RoboDK station: GenerischV4_OPCUA_cubestation.rdk

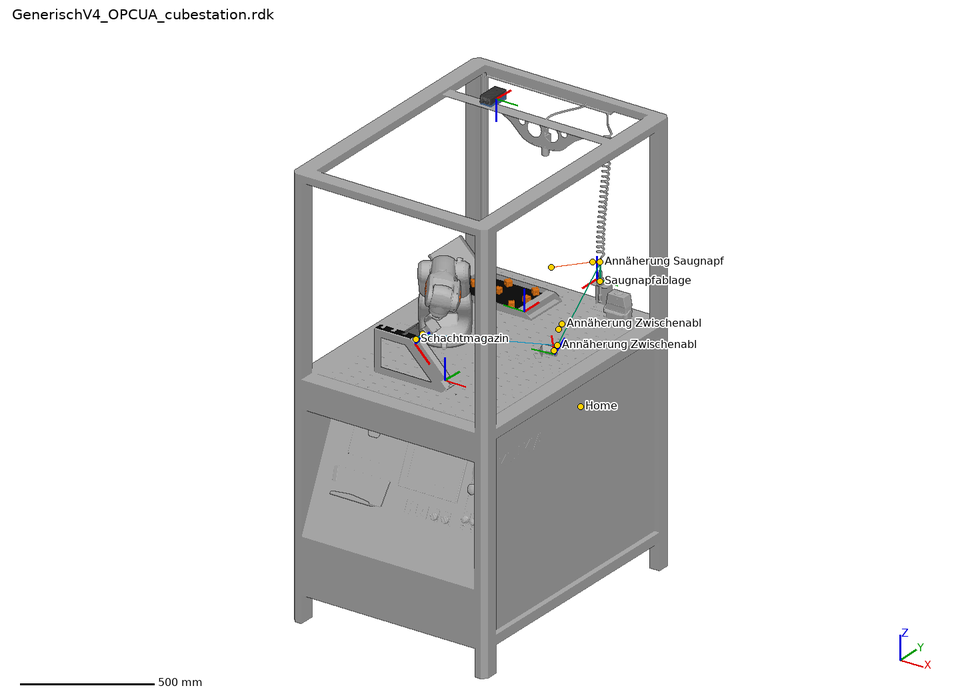
[picture v0: the station drawn from its stored meshes, robots at their saved joint values, targets as dots, program paths as lines]
Station GenerischV4_cubestation (saved by RoboDK 5.9.4). Poses are relative to the parent item; angles as X-Y-Z fixed-axis rotations.
Station parameters (name, value as stored): CMD_Objektposition, 0, CMD_Camera, 0, CMD_Annäherung_Saugnapf, 0, CMD_Aufraumen_Saugnapf, 0, CMD_Cube_1, 0, CMD_Cube_2, 0, CMD_Cube_3, 0, CMD_Cube_4, 0, CMD_Cube_5, 0, CMD_Cube_6, 0, CMD_Cube_7, 0, CMD_Cube_8, 0, CMD_Cube_9, 0, CMD_Main, 0, IO_1, 0, IO_2, 0, IO_3, 0, IO_4, 0, IO_5, 0, IO_6, 0, IO_7, 0, IO_8, 0, IO_9, 0, IO_10, 0, IO_11, 0, IO_12, 0, IO_13, 0, IO_14, 0, IO_15, 0, IO_16, 0, IO_17, 0, IO_18, 0, IO_19, 0, IO_20, 0, IO_21, 0, IO_22, 0, IO_23, 0, IO_24, 0, IO_25, 0, IO_26, 0, IO_27, 0, IO_28, 0, IO_29, 0, IO_30, 0, IO_31, 0, IO_32, 0, IO_33, 0, IO_34, 0, IO_35, 0, IO_36, 0, IO_37, 0, IO_38, 0, IO_39, 0, IO_40, 0, IO_41, 0, IO_42, 0, IO_43, 0, IO_44, 0, IO_45, 0, IO_46, 0, IO_47, 0, IO_48, 0, IO_49, 0, IO_50, 0, PY_RUNNING, 0, IO_Run, 0, CMD_SimulateCamera, 0, CMD_Annäherung_cube, 0, running, 0, OPC-UA, opc.tcp://localhost:4840
  - object Training_Cell at (0, 0, 166.87) mm, size 880 x 1200 x 1853 mm, geometry from Training_Cell_Ready2_educate_advanced.stl
  - frame KUKA KR 3 R540 Base at (0, 0, 0) mm
    - robot KUKA KR 3 R540: 6 axes, payload 3 kg, reach 541 mm, repeatability 0.02 mm, weight 26 kg
        modified DH rows (alpha deg, a mm, theta deg, d mm): 0, 0, 0, 345; -90, 20, 0, 0; 0, 260, -90, 0; -90, 20, 0, 260; 90, 0, 0, 0; -90, 0, 180, 75
        joint limits [-170, -170, -110, -175, -120, -350] to [170, 50, 155, 175, 120, 350]; home [0, -90, 90, 0, 0, 0]; saved at [56.786, -48.332, 48.725, 12.514, 97.773, 58.207]
      - tool Greifer, TCP at (38, 0, 110) mm, rotated rx 0 ry 30 rz 0 deg, size 63.3 x 66 x 118 mm
    - target Home (Cartesian target) at (549.5, 95.1, 7) mm, rotated rx 0 ry -90 rz -90.38 deg; joints [-2.455, -71.204, 142.326, -3.737, -41.152, -178.605] of KUKA KR 3 R540
  - frame Camera Reference at (-25, 370, 1007.5) mm, rotated rx -180 ry 0 rz 90 deg
    - object SICK VSPP-5F2113 at (0, 0, 0) mm, size 53 x 116 x 38 mm, geometry from SICK VSPx.sld
  - camera Kamera1
  - frame 9 wuerfelbett_t8_pxb7 at (152.39, 295.18, 209.01) mm, rotated rx 0.37 ry -0.77 rz 89.62 deg
    - object Cube 7 at (171.17, 70.32, -19.9) mm, rotated rx -0.78 ry 0.36 rz -39.63 deg, size 25 x 25 x 25 mm, geometry from Cube.stl
    - object Cube 8 at (101.17, 60.33, -18.89) mm, rotated rx -0.49 ry 0.7 rz -9.63 deg, size 25 x 25 x 25 mm, geometry from Cube.stl
    - object W at (8, 23, 3.2) mm, rotated rx -0.36 ry 0.77 rz 0.38 deg, size 200 x 470.5 x 147.4 mm, geometry from Deposit_2.stl
    - object Cube 9 at (100.63, 190.45, -19.73) mm, rotated rx -0.77 ry -0.37 rz -89.63 deg, size 25 x 25 x 25 mm, geometry from Cube.stl
    - object Cube 6 at (172.22, 194.56, -20.72) mm, rotated rx -0.7 ry 0.49 rz -29.63 deg, size 25 x 25 x 25 mm, geometry from Cube.stl
    - object Cube 5 at (173.17, 286.27, -21.32) mm, rotated rx -0.08 ry 0.85 rz 20.37 deg, size 25 x 25 x 25 mm, geometry from Cube.stl
    - object Cube 1 at (32.96, 83.65, -18.13) mm, rotated rx -0.22 ry -0.83 rz -139.62 deg, size 25 x 25 x 25 mm, geometry from Cube.stl
    - object Cube 2 at (49.33, 190.12, -19.04) mm, rotated rx -0.77 ry -0.37 rz -89.63 deg, size 25 x 25 x 25 mm, geometry from Cube.stl
    - object Cube 3 at (28.99, 289.92, -19.41) mm, rotated rx -0.23 ry 0.82 rz 10.37 deg, size 25 x 25 x 25 mm, geometry from Cube.stl
    - object Cube 4 at (99.32, 299.72, -20.42) mm, rotated rx -0.35 ry -0.78 rz -130 deg, size 25 x 25 x 25 mm, geometry from Cube.stl
  - frame 8  zwischenablage_t8_pxb7 at (427.29, 96.21, 189.23) mm, rotated rx 22.63 ry -21.63 rz 131.77 deg
    - object Zwischenablage at (44.58, 61.03, -55.36) mm, rotated rx 21.16 ry -23.07 rz 179.49 deg, size 94.7 x 93.8 x 35.5 mm, geometry from Deposit.stl
    - target Annäherung Zwischenablage 2 (Cartesian target) at (12.4, 2.45, 35.1) mm, rotated rx -180 ry 0 rz 0 deg; joints [-16.432, -24.429, 40.33, 17.251, 88.025, -57.396] of KUKA KR 3 R540
    - target Zwischenablage 2 (Cartesian target) at (12.4, 2.45, 5.1) mm, rotated rx 180 ry 0 rz 0 deg; joints [-16.926, -26.878, 50.942, 17.374, 80.369, -60.281] of KUKA KR 3 R540
  - frame 7 schachtmagazin_t8_pxb7 at (145, -402.24, 352.27) mm, rotated rx 0.31 ry 44.91 rz 0.8 deg
    - object Schachtmagazin at (-13.03, 7.5, -256.27) mm, rotated rx 0 ry -45 rz -0.8 deg, size 346.9 x 40 x 184.2 mm, geometry from Magazine.stl
    - target Annäherung Schachtmagazin (Cartesian target) at (-12, 23, 39) mm, rotated rx -180 ry 0 rz -180 deg; joints [56.786, -48.332, 48.725, 12.514, 97.773, 58.207] of KUKA KR 3 R540
    - target Schachtmagazin (Cartesian target) at (-12, 23, -1) mm, rotated rx -180 ry 0 rz 180 deg; joints [59.889, -52.448, 61.689, 12.835, 88.463, 59.286] of KUKA KR 3 R540
  - frame 10 werkzeugaufnahme_t8_pxb7 at (299.4, 557.1, 280) mm, rotated rx 0 ry 0 rz -90 deg
    - object werkzeugaufnahme at (505, -140, -1110) mm, rotated rx 0 ry 0 rz 90 deg, size 796 x 307.5 x 992.9 mm, geometry from Vaccumablage.stl
    - target Annäherung Saugnapf (Cartesian target) at (29.5, 35.1, 92) mm, rotated rx 0 ry -90 rz 0 deg; joints [-46.165, -35.886, 54.904, -65.833, 41.103, -95.129] of KUKA KR 3 R540
    - target Annäherung Würfelbetts (Cartesian target) at (155.64, -97.99, 83.31) mm, rotated rx 0 ry -90 rz 0 deg; joints [-47.815, -71.761, 116.568, 80.484, -36.134, -233.897] of KUKA KR 3 R540
    - target Annäherung Zwischenablage 1 (Cartesian target) at (457.77, 161.65, 41.46) mm, rotated rx 164.17 ry -60.61 rz 90.35 deg; joints [-23.461, -62.972, 94.422, 37.015, 42.384, -239.097] of KUKA KR 3 R540
    - target Zwischenablage 1 (Cartesian target) at (457.85, 146.24, 15.72) mm, rotated rx 164.17 ry -60.61 rz 90.35 deg; joints [-24.436, -62.797, 100.708, 42.078, 37.906, -246.437] of KUKA KR 3 R540
    - target Saugnapfablage (Cartesian target) at (29.5, 35.1, 12) mm, rotated rx 0 ry -90 rz 0 deg; joints [-46.165, -28.098, 58.876, -79.616, 37.574, -77.374] of KUKA KR 3 R540
    - target Federversatz (Cartesian target) at (79.5, 35.1, 112) mm, rotated rx 0 ry -90 rz 0 deg; joints [-41.734, -46.097, 68.534, -69.461, 43.641, -88.1] of KUKA KR 3 R540
    - object Saugnapf at (-1784, -698.7, 57.4) mm, rotated rx 180 ry 0 rz -90 deg, size 25.4 x 25 x 126.9 mm, geometry from Vacuum.stl
  - Python program SimulateCamera (listed below)
  - Python program Annäherung_cube (listed below)
  - program Objektposition (9 instructions, listed below)
  - program Camera (18 instructions, listed below)
  - program Annäherung_Saugnapf (12 instructions, listed below)
  - program Aufraumen_Saugnapf (13 instructions, listed below)
  - program Cube_1 (24 instructions, listed below)
  - program Cube_2 (24 instructions, listed below)
  - program Cube_3 (24 instructions, listed below)
  - program Cube_4 (24 instructions, listed below)
  - program Cube_5 (24 instructions, listed below)
  - program Cube_6 (24 instructions, listed below)
  - program Cube_7 (24 instructions, listed below)
  - program Cube_8 (24 instructions, listed below)
  - program Cube_9 (24 instructions, listed below)
  - program Main (36 instructions, listed below)
  - Python program Generisch4 (listed below)
  - Python program Generisch4_mit_zeit (listed below)
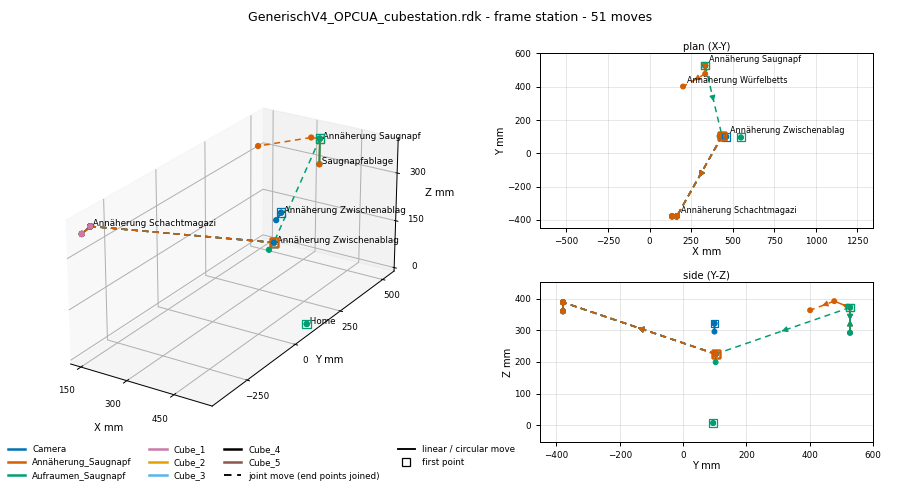
[picture p0: tool path of GenerischV4_OPCUA_cubestation.rdk in frame station, 51 of 51 moves have a stored position in this frame; points joined in program order, loops and branches not executed]

--- Python program SimulateCamera ---
from robolink import *
from robodk import *

RDK = Robolink()
while RDK.getParam("IO_15") !=1:
    time.sleep(0.05)
RDK.setParam("IO_Run", "1")

# --- Konfiguration von Roboter und Kamera ---
robot = RDK.Item('KUKA KR 3 R540', ITEM_TYPE_ROBOT)
frame_camera = RDK.Item('Camera Reference', ITEM_TYPE_FRAME)
base_name = "10 werkzeugaufnahme_t8_pxb7"
base_tool = RDK.Item('10 werkzeugaufnahme_t8_pxb7', ITEM_TYPE_FRAME)
robot.setPoseFrame(base_tool)
if not robot.Valid():
    raise Exception("Roboter nicht gefunden")
if not frame_camera.Valid():
    raise Exception("Kamera nicht gefunden")
if not base_tool.Valid():
    raise Exception("Werkzeugbasis nicht gefunden")

# Kamerapose in Basis 10
cam_in_base10 = invH(base_tool.PoseAbs()) * frame_camera.PoseAbs()

# --- Alle Würfel im Sichtfeld der Kamera erfassen ---
def get_detected_cubes_in_view(keyword='Cube'):
    detected = []
    all_objects = RDK.ItemList(ITEM_TYPE_OBJECT, True)
    for name in all_objects:
        if keyword in name:
            cube = RDK.Item(name)
            # Pose relativ zur Kamera
            pose_rel = invH(frame_camera.PoseAbs()) * cube.PoseAbs()
            tx, ty, tz, rx, ry, rz = pose_2_xyzrpw(pose_rel)
            # Filterung nach Sichtfeld (Grenzen je nach Kamera anpassen)
            if -200 <= tx <= 200 and -200 <= ty <= 200 and 0 <= tz <= 1000:
                detected.append(name)
    detected.sort()  # Alphabetische Sortierung: Cube 1, Cube 2 ...
    print(f"Im Sichtfeld erkannte Würfel: {detected} (insgesamt {len(detected)})")
    return detected

# --- Auswahl des Würfels (immer der kleinste sichtbare) ---
def choose_cube(detected_cubes):
    if not detected_cubes:
        raise Exception("Keine Würfel im Sichtfeld der Kamera")
    return detected_cubes[0]

# --- Pose des Würfels in Basis 10 bestimmen ---
def detect_cube_pose(cube_name):
    all_objects = RDK.ItemList(ITEM_TYPE_OBJECT, True)
    for name in all_objects:
        if cube_name == name:
            cube = RDK.Item(name)
            pose_rel = invH(frame_camera.PoseAbs()) * cube.PoseAbs()
            return cam_in_base10 * transl(pose_rel[0,3], pose_rel[1,3], pose_rel[2,3])
    raise Exception(f"{cube_name} nicht gefunden")

# --- Hauptprogramm ---
detected_cubes = get_detected_cubes_in_view()
cube_to_pick = choose_cube(detected_cubes)
cube_pose = detect_cube_pose(cube_to_pick)

# XY-Ausrichtung des Roboters
current_pose = robot.Pose()
aligned_pose = current_pose.copy()
aligned_pose[0,3] = cube_pose[0,3]
aligned_pose[1,3] = cube_pose[1,3]
robot.MoveL(aligned_pose)
print(f"Roboter XY ausgerichtet mit {cube_to_pick}")

# Absenken für Greiferbefestigung
grasp_pose = aligned_pose.copy()
grasp_pose[2,3] = 18.400
robot.MoveL(grasp_pose)
print(f"Roboter abgesenkt zum Greiferanbringen für {cube_to_pick}")

RDK.setParam("IO_Run", "0")
RDK.setParam("running", "0")
RDK.setParam("IO_15", "0")

--- Python program Annäherung_cube ---
from robolink import *
from robodk import *

RDK = Robolink()
while RDK.getParam("IO_16") !=1:
    time.sleep(0.05)
RDK.setParam("IO_Run", "1")
# Roboter und Werkzeugbasis
robot = RDK.Item('KUKA KR 3 R540', ITEM_TYPE_ROBOT)
base_tool = RDK.Item('10 werkzeugaufnahme_t8_pxb7', ITEM_TYPE_FRAME)

if not robot.Valid():
    raise Exception("Roboter nicht gefunden")
if not base_tool.Valid():
    raise Exception("Werkzeugbasis nicht gefunden")

# Aktuelle Pose des Roboters
current_pose = robot.Pose()

# Z-Movement auf 68.400 in Basis 10
target_pose = current_pose.copy()
target_pose[2,3] = 68.400

robot.MoveL(target_pose)
print("Roboter auf Z=68.400 angehoben")
RDK.setParam("IO_Run", "0")
RDK.setParam("running", "0")
RDK.setParam("IO_16", "0")

--- program Objektposition (robot KUKA KR 3 R540) ---
  Wait IO_1=1
  Set IO_Run=1
  Remplacer Saugnapf
  Replacer Würfel 1
  Replacer Würfel 2
  Replacer Würfel 3
  Replacer objets
  Set IO_Run=0
  Set IO_1=0

--- program Camera (robot KUKA KR 3 R540) ---
  Wait IO_2=1
  Set IO_Run=1
  Définir Ref.: 10 werkzeugaufnahme_t8_pxb7
  Choisir Outil: Greifer
  Set IO_15=1
  Call SimulateCamera
  Set IO_Run=1
  Attach to Greifer
  Set IO_16=1
  Call Annäherung_cube
  Set IO_Run=1
  MoveJ (Annäherung Zwischenablage 1)
  MoveL (Zwischenablage 1)
  Detach from Greifer
  Attach to Greifer
  MoveL (Annäherung Zwischenablage) -> target Annäherung Zwischenablage 1
  Set IO_Run=0
  Set IO_2=0

--- program Annäherung_Saugnapf (robot KUKA KR 3 R540) ---
  Wait IO_3=1
  Set IO_Run=1
  Définir Ref.: 10 werkzeugaufnahme_t8_pxb7
  Choisir Outil: Greifer
  MoveJ (Annäherung Saugnapf)
  MoveL (Saugnapfablage)
  Attacher à Greifer
  MoveL (Annäherung Saugnapf)
  MoveL (Federversatz)
  MoveJ (Annäherung Würfelbetts)
  Set IO_Run=0
  Set IO_3=0

--- program Aufraumen_Saugnapf (robot KUKA KR 3 R540) ---
  Wait IO_4=1
  Set IO_Run=1
  Définir Ref.: 10 werkzeugaufnahme_t8_pxb7
  Choisir Outil: Greifer
  MoveJ (Annäherung Saugnapf)
  MoveL (Saugnapfablage)
  Détachez de Greifer
  MoveL (Annäherung Saugnapf)
  Définir Ref.: Frame_Deposit -> 8  zwischenablage_t8_pxb7
  MoveJ (Annäherung Zwischenablage 2)
  MoveL (Zwischenablage 2)
  Set IO_Run=0
  Set IO_4=0

--- program Cube_1 (robot KUKA KR 3 R540) ---
  Wait IO_5=1
  Set IO_Run=1
  Set Ref.: 10 werkzeugaufnahme_t8_pxb7
  Set Tool: Greifer
  Set IO_3=1
  Call Annäherung_Saugnapf
  Set IO_Run=1
  Set IO_2=1
  Call Camera
  Set IO_Run=1
  Replace Cube 1
  Set IO_4=1
  Call Aufraumen_Saugnapf
  Set IO_Run=1
  Attach to Greifer
  MoveL (Annäherung Zwischenablage) -> target Annäherung Zwischenablage 2
  Set Ref.: 7 schachtmagazin_t8_pxb7
  MoveJ (Annäherung Schachtmagazin)
  MoveL (Schachtmagazin)
  Detach from Greifer
  MoveL (Annäherung Schachtmagazin)
  Replace Cube 1
  Set IO_Run=0
  Set IO_5=0

--- program Cube_2 (robot KUKA KR 3 R540) ---
  Wait IO_6=1
  Set IO_Run=1
  Définir Ref.: 10 werkzeugaufnahme_t8_pxb7
  Choisir Outil: Greifer
  Set IO_3=1
  Appel Annäherung_Saugnapf
  Set IO_Run=1
  Set IO_2=1
  Appel Camera
  Set IO_Run=1
  Remplacer Cube 2
  Set IO_4=1
  Appel Aufraumen_Saugnapf
  Set IO_Run=1
  Attacher à Greifer
  MoveL (Annäherung Zwischenablage) -> target Annäherung Zwischenablage 2
  Définir Ref.: 7 schachtmagazin_t8_pxb7
  MoveJ (Annäherung Schachtmagazin)
  MoveL (Schachtmagazin)
  Détachez de Greifer
  MoveL (Annäherung Schachtmagazin)
  Remplacer Cube 2
  Set IO_Run=0
  Set IO_6=0

--- program Cube_3 (robot KUKA KR 3 R540) ---
  Wait IO_7=1
  Set IO_Run=1
  Définir Ref.: 10 werkzeugaufnahme_t8_pxb7
  Choisir Outil: Greifer
  Set IO_3=1
  Appel Annäherung_Saugnapf
  Set IO_Run=1
  Set IO_2=1
  Appel Camera
  Set IO_Run=1
  Remplacer Cube 3
  Set IO_4=1
  Appel Aufraumen_Saugnapf
  Set IO_Run=1
  Attacher à Greifer
  MoveL (Annäherung Zwischenablage) -> target Annäherung Zwischenablage 2
  Définir Ref.: 7 schachtmagazin_t8_pxb7
  MoveJ (Annäherung Schachtmagazin)
  MoveL (Schachtmagazin)
  Détachez de Greifer
  MoveL (Annäherung Schachtmagazin)
  Remplacer Cube 3
  Set IO_Run=0
  Set IO_7=0

--- program Cube_4 (robot KUKA KR 3 R540) ---
  Wait IO_8=1
  Set IO_Run=1
  Définir Ref.: 10 werkzeugaufnahme_t8_pxb7
  Choisir Outil: Greifer
  Set IO_3=1
  Appel Annäherung_Saugnapf
  Set IO_Run=1
  Set IO_2=1
  Appel Camera
  Set IO_Run=1
  Remplacer Cube 4
  Set IO_4=1
  Appel Aufraumen_Saugnapf
  Set IO_Run=1
  Attacher à Greifer
  MoveL (Annäherung Zwischenablage) -> target Annäherung Zwischenablage 2
  Définir Ref.: 7 schachtmagazin_t8_pxb7
  MoveJ (Annäherung Schachtmagazin)
  MoveL (Schachtmagazin)
  Détachez de Greifer
  MoveL (Annäherung Schachtmagazin)
  Remplacer Cube 4
  Set IO_Run=0
  Set IO_8=0

--- program Cube_5 (robot KUKA KR 3 R540) ---
  Wait IO_9=1
  Set IO_Run=1
  Définir Ref.: 10 werkzeugaufnahme_t8_pxb7
  Choisir Outil: Greifer
  Set IO_3=1
  Appel Annäherung_Saugnapf
  Set IO_Run=1
  Set IO_2=1
  Appel Camera
  Set IO_Run=1
  Remplacer Cube 5
  Set IO_4=1
  Appel Aufraumen_Saugnapf
  Set IO_Run=1
  Attacher à Greifer
  MoveL (Annäherung Zwischenablage) -> target Annäherung Zwischenablage 2
  Définir Ref.: 7 schachtmagazin_t8_pxb7
  MoveJ (Annäherung Schachtmagazin)
  MoveL (Schachtmagazin)
  Détachez de Greifer
  MoveL (Annäherung Schachtmagazin)
  Remplacer Cube 5
  Set IO_Run=0
  Set IO_9=0

--- program Cube_6 (robot KUKA KR 3 R540) ---
  Wait IO_10=1
  Set IO_Run=1
  Définir Ref.: 10 werkzeugaufnahme_t8_pxb7
  Choisir Outil: Greifer
  Set IO_3=1
  Appel Annäherung_Saugnapf
  Set IO_Run=1
  Set IO_2=1
  Appel Camera
  Set IO_Run=1
  Remplacer Cube 6
  Set IO_4=1
  Appel Aufraumen_Saugnapf
  Set IO_Run=1
  Attacher à Greifer
  MoveL (Annäherung Zwischenablage) -> target Annäherung Zwischenablage 2
  Définir Ref.: 7 schachtmagazin_t8_pxb7
  MoveJ (Annäherung Schachtmagazin)
  MoveL (Schachtmagazin)
  Détachez de Greifer
  MoveL (Annäherung Schachtmagazin)
  Remplacer Cube 6
  Set IO_Run=0
  Set IO_10=0

--- program Cube_7 (robot KUKA KR 3 R540) ---
  Wait IO_11=1
  Set IO_Run=1
  Définir Ref.: 10 werkzeugaufnahme_t8_pxb7
  Choisir Outil: Greifer
  Set IO_3=1
  Appel Annäherung_Saugnapf
  Set IO_Run=1
  Set IO_2=1
  Appel Camera
  Set IO_Run=1
  Remplacer Cube 7
  Set IO_4=1
  Appel Aufraumen_Saugnapf
  Set IO_Run=1
  Attacher à Greifer
  MoveL (Annäherung Zwischenablage) -> target Annäherung Zwischenablage 2
  Définir Ref.: 7 schachtmagazin_t8_pxb7
  MoveJ (Annäherung Schachtmagazin)
  MoveL (Schachtmagazin)
  Détachez de Greifer
  MoveL (Annäherung Schachtmagazin)
  Remplacer Cube 7
  Set IO_Run=0
  Set IO_11=0

--- program Cube_8 (robot KUKA KR 3 R540) ---
  Wait IO_12=1
  Set IO_Run=1
  Définir Ref.: 10 werkzeugaufnahme_t8_pxb7
  Choisir Outil: Greifer
  Set IO_3=1
  Appel Annäherung_Saugnapf
  Set IO_Run=1
  Set IO_2=1
  Appel Camera
  Set IO_Run=1
  Remplacer Cube 8
  Set IO_4=1
  Appel Aufraumen_Saugnapf
  Set IO_Run=1
  Attacher à Greifer
  MoveL (Annäherung Zwischenablage) -> target Annäherung Zwischenablage 2
  Définir Ref.: 7 schachtmagazin_t8_pxb7
  MoveJ (Annäherung Schachtmagazin)
  MoveL (Schachtmagazin)
  Détachez de Greifer
  MoveL (Annäherung Schachtmagazin)
  Remplacer Cube 8
  Set IO_Run=0
  Set IO_12=0

--- program Cube_9 (robot KUKA KR 3 R540) ---
  Wait IO_13=1
  Set IO_Run=1
  Définir Ref.: 10 werkzeugaufnahme_t8_pxb7
  Choisir Outil: Greifer
  Set IO_3=1
  Appel Annäherung_Saugnapf
  Set IO_Run=1
  Set IO_2=1
  Appel Camera
  Set IO_Run=1
  Remplacer Cube 9
  Set IO_4=1
  Appel Aufraumen_Saugnapf
  Set IO_Run=1
  Attacher à Greifer
  MoveL (Annäherung Zwischenablage) -> target Annäherung Zwischenablage 2
  Définir Ref.: 7 schachtmagazin_t8_pxb7
  MoveJ (Annäherung Schachtmagazin)
  MoveL (Schachtmagazin)
  Détachez de Greifer
  MoveL (Annäherung Schachtmagazin)
  Remplacer Cube 9
  Set IO_Run=0
  Set IO_13=0

--- program Main (robot KUKA KR 3 R540) ---
  Wait IO_14=1
  Set IO_Run=1
  Définir Ref.: 10 werkzeugaufnahme_t8_pxb7
  Choisir Outil: Greifer
  MoveJ (Home)
  Set IO_5=1
  Appel Cube_1
  Set IO_Run=1
  Set IO_6=1
  Appel Cube_2
  Set IO_Run=1
  Set IO_7=1
  Appel Cube_3
  Set IO_Run=1
  Set IO_8=1
  Appel Cube_4
  Set IO_Run=1
  Set IO_9=1
  Appel Cube_5
  Set IO_Run=1
  Set IO_10=1
  Appel Cube_6
  Set IO_Run=1
  Set IO_11=1
  Appel Cube_7
  Set IO_Run=1
  Set IO_12=1
  Appel Cube_8
  Set IO_Run=1
  Set IO_13=1
  Appel Cube_9
  Set IO_Run=1
  Définir Ref.: 10 werkzeugaufnahme_t8_pxb7
  MoveJ (Home)
  Set IO_Run=0
  Set IO_14=0

--- Python program Generisch4 ---
from robodk import robolink
from robodk.robolink import ITEM_TYPE_PROGRAM, ITEM_TYPE_PROGRAM_PYTHON
from opcua import Client, ua
import time

print("=== START ROBOdk / OPC-UA SCRIPT ===")

# ============================================================
# RoboDK Verbindung
# ------------------------------------------------------------
# Aufbau der Verbindung zur aktuell geöffneten RoboDK-Station.
# Über diese Schnittstelle werden Programme gestartet,
# Parameter gelesen/geschrieben und IO-Zustände abgefragt.
# ============================================================
RDK = robolink.Robolink()

# ============================================================
# OPC-UA Verbindung (CODESYS PLC)
# ------------------------------------------------------------
# Verbindung zum OPC-UA Server der CODESYS Runtime.
# Dieser Server stellt alle PLC-Variablen zur Verfügung,
# die für die Kommunikation mit RoboDK benötigt werden.
# ============================================================
client = Client("opc.tcp://localhost:4840")
client.connect()
print("OPC-UA connected")

# ============================================================
# OPC-UA Nodes (PLC Variablen)
# ------------------------------------------------------------
# Alle relevanten PLC-Variablen werden hier einmalig
# über ihren Node-Pfad referenziert.
# ============================================================
node_names   = client.get_node("ns=4;s=|var|CODESYS Control Win V3 x64.Application.GVL.Comb_names")
node_nb      = client.get_node("ns=4;s=|var|CODESYS Control Win V3 x64.Application.GVL.Nb_Programs")
node_sel     = client.get_node("ns=4;s=|var|CODESYS Control Win V3 x64.Application.GVL.Selected_Index")
node_trigger = client.get_node("ns=4;s=|var|CODESYS Control Win V3 x64.Application.GVL.Trigger")
node_stop    = client.get_node("ns=4;s=|var|CODESYS Control Win V3 x64.Application.GVL.Stop")

# IO-Befehle vom PLC (Start-IOs)
node_io_cmd  = client.get_node("ns=4;s=|var|CODESYS Control Win V3 x64.Application.GVL.IO_")

# Rückmeldung: Programm läuft (echter Status aus RoboDK)
node_io_run  = client.get_node("ns=4;s=|var|CODESYS Control Win V3 x64.Application.GVL.IO_Run")

# Aktuell ausgeführtes Programm
node_cur     = client.get_node("ns=4;s=|var|CODESYS Control Win V3 x64.Application.GVL.Current_Program")

# ============================================================
# Konstanten
# ------------------------------------------------------------
# Maximale Anzahl unterstützter Programme / IOs
# ============================================================
MAX = 50

# ============================================================
# Interne Zustände (nur im Python-Skript)
# ------------------------------------------------------------
# Diese Variablen dienen zur sauberen Flankenerkennung
# und zur internen Ablaufsteuerung.
# ============================================================
prev_trigger = False                    # Trigger-Flankenerkennung
prev_io_cmd = [False] * MAX             # IO-Flankenerkennung

program_running = False                 # interner Laufstatus
current_program_item = None             # aktuelles RoboDK-Programmobjekt
current_program_is_python = False       # Programmart (Standard / Python)

# ============================================================
# Initialisierung
# ------------------------------------------------------------
# Alle IOs werden beim Start explizit auf 0 gesetzt,
# um einen definierten Anfangszustand sicherzustellen.
# ============================================================
for i in range(1, MAX + 1):
    RDK.setParam(f"IO_{i}", "0")

# ============================================================
# Hauptschleife
# ------------------------------------------------------------
# Zyklische Verarbeitung:
# - Programmliste aktualisieren
# - PLC-Eingänge auswerten
# - IOs synchronisieren
# - Programme starten / stoppen
# ============================================================
while True:
    try:
        # ====================================================
        # Programmliste aus RoboDK lesen
        # ----------------------------------------------------
        # Alle Programme, die mit "CMD_" beginnen, werden
        # als steuerbare Programme betrachtet.
        # ====================================================
        params = RDK.getParams()
        cmd_programs = [n for n, v in params if n.startswith("CMD_")]

        names = cmd_programs + [""] * (MAX - len(cmd_programs))
        node_names.set_value(ua.Variant(names, ua.VariantType.String))
        node_nb.set_value(ua.Variant(len(cmd_programs), ua.VariantType.Int16))

        # ====================================================
        # PLC Variablen lesen
        # ====================================================
        sel = node_sel.get_value()
        trigger = node_trigger.get_value()
        stop_cmd = node_stop.get_value()
        io_cmd = list(node_io_cmd.get_value())

        # ====================================================
        # PLC → RoboDK : IO_n (nur steigende Flanke)
        # ----------------------------------------------------
        # Dadurch wird verhindert, dass IOs zyklisch
        # überschrieben oder mehrfach gesetzt werden.
        # ====================================================
        for i in range(1, MAX + 1):
            plc_val = bool(io_cmd[i - 1])

            if plc_val and not prev_io_cmd[i - 1]:
                print(f"[PLC→RDK] Rising edge IO_{i}")
                RDK.setParam(f"IO_{i}", "1")

            prev_io_cmd[i - 1] = plc_val

        # ====================================================
        # RoboDK → PLC : IO Feedback
        # ----------------------------------------------------
        # Der echte IO-Zustand aus RoboDK wird zurück
        # an das PLC gemeldet (kein virtuelles Feedback).
        # ====================================================
        io_feedback = [False] * MAX

        for i in range(1, MAX + 1):
            val = RDK.getParam(f"IO_{i}")
            try:
                io_feedback[i - 1] = bool(int(val))
            except:
                io_feedback[i - 1] = False

        node_io_cmd.set_value(ua.Variant(io_feedback, ua.VariantType.Boolean))

        # ====================================================
        # IO_Run
        # ----------------------------------------------------
        # IO_Run wird ausschließlich von den RoboDK-
        # Programmen selbst gesetzt (Standard & Python).
        # Dieses Skript liest den Zustand nur aus.
        # ====================================================
        io_run_raw = RDK.getParam("IO_Run")
        io_run = bool(int(io_run_raw)) if io_run_raw else False
        node_io_run.set_value(io_run)

        # ====================================================
        # STOP-Befehl vom PLC
        # ====================================================
        if stop_cmd:
            print("STOP empfangen")

            try:
                if current_program_item and current_program_item.Valid():
                    current_program_item.Stop()
            except:
                pass

            # Alle IOs zurücksetzen
            for i in range(1, MAX + 1):
                RDK.setParam(f"IO_{i}", "0")

            RDK.setParam("IO_Run", "0")

            node_io_cmd.set_value(ua.Variant([False] * MAX, ua.VariantType.Boolean))
            node_cur.set_value("")
            node_stop.set_value(False)

            program_running = False
            current_program_item = None
            current_program_is_python = False

        # ====================================================
        # START-Befehl
        # ====================================================
        if trigger and not prev_trigger and not program_running:
            if 1 <= sel <= len(cmd_programs):
                prog_name = names[sel - 1].replace("CMD_", "")

                prog = RDK.Item(prog_name)
                if not prog.Valid():
                    raise Exception("RoboDK Programm nicht gefunden")

                # Aktuelles Programm im PLC anzeigen
                node_cur.set_value(prog_name)
                print(prog_name)

                if prog.Type() == ITEM_TYPE_PROGRAM_PYTHON:
                    current_program_is_python = True
                    RDK.setParam("running", "1")
                    RDK.RunCode(prog_name)
                else:
                    current_program_is_python = False
                    prog.RunProgram()

                program_running = True
                current_program_item = prog
                node_trigger.set_value(False)

        prev_trigger = trigger

        # ====================================================
        # Programmen­de erkennen
        # ====================================================
        if program_running:
            if current_program_is_python:
                io_running = RDK.getParam("running")
                finished = not bool(int(io_running)) if io_running else True
            else:
                finished = not current_program_item.Busy()

            if finished:
                print("Programm beendet")

                program_running = False
                current_program_item = None
                current_program_is_python = False
                node_cur.set_value("")

        time.sleep(0.09)


    except Exception as e:
        print("FEHLER:", e)
        time.sleep(0.5)

--- Python program Generisch4_mit_zeit ---
from robodk import robolink
from robodk.robolink import ITEM_TYPE_PROGRAM, ITEM_TYPE_PROGRAM_PYTHON
from opcua import Client, ua
import time

print("=== START ROBOdk / OPC-UA SCRIPT ===")

# ============================================================
# RoboDK Verbindung
# ------------------------------------------------------------
# Aufbau der Verbindung zur aktuell geöffneten RoboDK-Station.
# Über diese Schnittstelle werden Programme gestartet,
# Parameter gelesen/geschrieben und IO-Zustände abgefragt.
# ============================================================
RDK = robolink.Robolink()

# ============================================================
# OPC-UA Verbindung (CODESYS PLC)
# ------------------------------------------------------------
# Verbindung zum OPC-UA Server der CODESYS Runtime.
# Dieser Server stellt alle PLC-Variablen zur Verfügung,
# die für die Kommunikation mit RoboDK benötigt werden.
# ============================================================
client = Client("opc.tcp://localhost:4840")
client.connect()
print("OPC-UA connected")

# ============================================================
# OPC-UA Nodes (PLC Variablen)
# ------------------------------------------------------------
# Alle relevanten PLC-Variablen werden hier einmalig
# über ihren Node-Pfad referenziert.
# ============================================================
node_names   = client.get_node("ns=4;s=|var|CODESYS Control Win V3 x64.Application.GVL.Comb_names")
node_nb      = client.get_node("ns=4;s=|var|CODESYS Control Win V3 x64.Application.GVL.Nb_Programs")
node_sel     = client.get_node("ns=4;s=|var|CODESYS Control Win V3 x64.Application.GVL.Selected_Index")
node_trigger = client.get_node("ns=4;s=|var|CODESYS Control Win V3 x64.Application.GVL.Trigger")
node_stop    = client.get_node("ns=4;s=|var|CODESYS Control Win V3 x64.Application.GVL.Stop")

# IO-Befehle vom PLC (Start-IOs)
node_io_cmd  = client.get_node("ns=4;s=|var|CODESYS Control Win V3 x64.Application.GVL.IO_")

# Rückmeldung: Programm läuft (echter Status aus RoboDK)
node_io_run  = client.get_node("ns=4;s=|var|CODESYS Control Win V3 x64.Application.GVL.IO_Run")

# Aktuell ausgeführtes Programm
node_cur     = client.get_node("ns=4;s=|var|CODESYS Control Win V3 x64.Application.GVL.Current_Program")

# ============================================================
# Konstanten
# ------------------------------------------------------------
# Maximale Anzahl unterstützter Programme / IOs
# ============================================================
MAX = 50

# ============================================================
# Interne Zustände (nur im Python-Skript)
# ------------------------------------------------------------
# Diese Variablen dienen zur sauberen Flankenerkennung
# und zur internen Ablaufsteuerung.
# ============================================================
prev_trigger = False                    # Trigger-Flankenerkennung
prev_io_cmd = [False] * MAX             # IO-Flankenerkennung

program_running = False                 # interner Laufstatus
current_program_item = None             # aktuelles RoboDK-Programmobjekt
current_program_is_python = False       # Programmart (Standard / Python)

# ============================================================
# Initialisierung
# ------------------------------------------------------------
# Alle IOs werden beim Start explizit auf 0 gesetzt,
# um einen definierten Anfangszustand sicherzustellen.
# ============================================================
for i in range(1, MAX + 1):
    RDK.setParam(f"IO_{i}", "0")

# ============================================================
# Hauptschleife
# ------------------------------------------------------------
# Zyklische Verarbeitung:
# - Programmliste aktualisieren
# - PLC-Eingänge auswerten
# - IOs synchronisieren
# - Programme starten / stoppen
# ============================================================
while True:
    Start = time.perf_counter() # Startet einen hochpräzisen Zähler
    try:
        # ====================================================
        # Programmliste aus RoboDK lesen
        # ----------------------------------------------------
        # Alle Programme, die mit "CMD_" beginnen, werden
        # als steuerbare Programme betrachtet.
        # ====================================================
        params = RDK.getParams()
        cmd_programs = [n for n, v in params if n.startswith("CMD_")]

        names = cmd_programs + [""] * (MAX - len(cmd_programs))
        node_names.set_value(ua.Variant(names, ua.VariantType.String))
        node_nb.set_value(ua.Variant(len(cmd_programs), ua.VariantType.Int16))

        # ====================================================
        # PLC Variablen lesen
        # ====================================================
        sel = node_sel.get_value()
        trigger = node_trigger.get_value()
        stop_cmd = node_stop.get_value()
        io_cmd = list(node_io_cmd.get_value())

        # ====================================================
        # PLC → RoboDK : IO_n (nur steigende Flanke)
        # ----------------------------------------------------
        # Dadurch wird verhindert, dass IOs zyklisch
        # überschrieben oder mehrfach gesetzt werden.
        # ====================================================
        for i in range(1, MAX + 1):
            plc_val = bool(io_cmd[i - 1])

            if plc_val and not prev_io_cmd[i - 1]:
                print(f"[PLC→RDK] Rising edge IO_{i}")
                RDK.setParam(f"IO_{i}", "1")

            prev_io_cmd[i - 1] = plc_val

        # ====================================================
        # RoboDK → PLC : IO Feedback
        # ----------------------------------------------------
        # Der echte IO-Zustand aus RoboDK wird zurück
        # an das PLC gemeldet (kein virtuelles Feedback).
        # ====================================================
        io_feedback = [False] * MAX

        for i in range(1, MAX + 1):
            val = RDK.getParam(f"IO_{i}")
            try:
                io_feedback[i - 1] = bool(int(val))
            except:
                io_feedback[i - 1] = False

        node_io_cmd.set_value(ua.Variant(io_feedback, ua.VariantType.Boolean))

        # ====================================================
        # IO_Run
        # ----------------------------------------------------
        # IO_Run wird ausschließlich von den RoboDK-
        # Programmen selbst gesetzt (Standard & Python).
        # Dieses Skript liest den Zustand nur aus.
        # ====================================================
        io_run_raw = RDK.getParam("IO_Run")
        io_run = bool(int(io_run_raw)) if io_run_raw else False
        node_io_run.set_value(io_run)

        # ====================================================
        # STOP-Befehl vom PLC
        # ====================================================
        if stop_cmd:
            print("STOP empfangen")

            try:
                if current_program_item and current_program_item.Valid():
                    current_program_item.Stop()
            except:
                pass

            # Alle IOs zurücksetzen
            for i in range(1, MAX + 1):
                RDK.setParam(f"IO_{i}", "0")

            RDK.setParam("IO_Run", "0")

            node_io_cmd.set_value(ua.Variant([False] * MAX, ua.VariantType.Boolean))
            node_cur.set_value("")
            node_stop.set_value(False)

            program_running = False
            current_program_item = None
            current_program_is_python = False

        # ====================================================
        # START-Befehl
        # ====================================================
        if trigger and not prev_trigger and not program_running:
            if 1 <= sel <= len(cmd_programs):
                prog_name = names[sel - 1].replace("CMD_", "")

                prog = RDK.Item(prog_name)
                if not prog.Valid():
                    raise Exception("RoboDK Programm nicht gefunden")

                # Aktuelles Programm im PLC anzeigen
                node_cur.set_value(prog_name)
                print(prog_name)

                if prog.Type() == ITEM_TYPE_PROGRAM_PYTHON:
                    current_program_is_python = True
                    RDK.setParam("running", "1")
                    RDK.RunCode(prog_name)
                else:
                    current_program_is_python = False
                    prog.RunProgram()

                program_running = True
                current_program_item = prog
                node_trigger.set_value(False)

        prev_trigger = trigger

        # ====================================================
        # Programmen­de erkennen
        # ====================================================
        if program_running:
            if current_program_is_python:
                io_running = RDK.getParam("running")
                finished = not bool(int(io_running)) if io_running else True
            else:
                finished = not current_program_item.Busy()

            if finished:
                print("Programm beendet")

                program_running = False
                current_program_item = None
                current_program_is_python = False
                node_cur.set_value("")

        time.sleep(0.09)
        end = time.perf_counter() # Stoppen Sie den Zähler
        print(f"Verstrichene Zeit : {end - Start:.3f} Sekunden")


    except Exception as e:
        print("FEHLER:", e)
        time.sleep(0.5)
